(* PLC project Untitled1, Beckhoff Automation GmbH TF6420 Database Server Query Analyser 1.0.0.0 *)
(* stored: creationDateTime 2026-03-11T15:45:14, modificationDateTime 2026-03-11T15:45:14 *)

TYPE ST_VALORES : STRUCT
  id : DINT;
  nome : STRING(30);
  valor : REAL;
END_STRUCT;
END_TYPE
